FUNCTION_BLOCK InfluxMessage
VAR_INPUT
	// payload string received
	sPayload:	STRING(255);
END_VAR
VAR_OUTPUT
	// measurement string (first word)
	measurement:	STRING(255) := '';
	// parameter (variable name)
	parameter:		STRING(255) := '';
	// value (variable content)
	value:			STRING(255) := '';
END_VAR
VAR
	space_position:		INT;
	equial_position:	INT;
	comma_position:		INT;
	measurement_tags:	STRING(255);
	parameter_value: 	STRING(255);
	bResultSplit: 		BOOL;
	// definition of the space separator
	spaceSeparator:		STRING(1) := ' ';
	// definition of the comma separator
	commaSeparator:		STRING(1) := ',';
	// definition of the equial sign separator
	equialSeparator:	STRING(1) := '=';
END_VAR

(* 
parse message in influx format:
	measurement parameter=value
	measurement,tag1=tag1value parameter=value

Multiple parameter/value pairs are ignored for now.
tags are not supported.
*)

//separate measurement from parameter, value
bResultSplit := FindAndSplit( pSeparator     := ADR(spaceSeparator), pSrcString := ADR(sPayload), 
                              pLeftString    := ADR(measurement_tags), nLeftSize  := SIZEOF(measurement_tags), 
                              pRightString   := ADR(parameter_value), nRightSize := SIZEOF(parameter_value),
                              bSearchFromRight := FALSE );
IF NOT bResultSplit THEN
	RETURN;
END_IF
// look for tags attached to the measurement
comma_position := FIND(measurement_tags, commaSeparator);
IF comma_position = 0 THEN
	measurement := measurement_tags;
ELSE
	measurement := LEFT(measurement_tags, comma_position-1);
END_IF
// dissect the parameter=value part
bResultSplit := FindAndSplit( pSeparator     := ADR(equialSeparator), pSrcString := ADR(parameter_value), 
                              pLeftString    := ADR(parameter), nLeftSize  := SIZEOF(parameter), 
                              pRightString   := ADR(value), nRightSize := SIZEOF(value),
                              bSearchFromRight := FALSE );

END_FUNCTION_BLOCK

(* stored: Version 1.1.0.1, ProductVersion 3.1.4024.9
   POU InfluxMessage: Id {90ca1cc6-8109-4bcf-9f8e-c5cf65cdb4b2}, SpecialFunc None *)
